# B&R Automation Studio project lab1_SFMRS
Automation Studio 

## Logical view

### Program Logical/MotorContr

#### FB_Integrator.c
```c
#include <bur/plctypes.h>
#ifdef __cplusplus
	extern "C"
	{
#endif
	#include "MotorContr.h"
#ifdef __cplusplus
	};
#endif
/* intrigal */
void FB_Integrator(struct FB_Integrator* inst)
{
	inst->dt=0.02;
	inst->out = inst->dt * inst->in + inst->state;
	inst->state = inst->out;

}
```

#### FB_motor.c
```c
#include <bur/plctypes.h>
#ifdef __cplusplus
	extern "C"
	{
#endif
	#include "MotorContr.h"
#ifdef __cplusplus
	};
#endif
/* FB motorrrrrrrrrrrrrrrrrrrrrrrrr */
void FB_motor(struct FB_motor* inst)
{
	REAL signal_1 = (inst->u) / inst->ke - inst->w;
	REAL signal_2 = signal_1 / inst->Tm;

	inst->w_integrator.in = signal_2;
	FB_Integrator(&inst->w_integrator);
	inst->w = inst->w_integrator.out;

	inst->phi_integrator.in = inst->w;
	FB_Integrator(&inst->phi_integrator);
	inst->phi = inst->phi_integrator.out;
}
```

### Variables.var
```iecst
VAR
	speed : REAL;
	enable : BOOL := TRUE;
	fb_regulator : FB_regulator;
	fb_motor : FB_motor;
	fb_motor2 : FB_motor;
	counter : INT;
	cnt2 : INT;
END_VAR
```
